TYPE ST_CX_NVDataBlock :
STRUCT
	DataOffs	: UDINT;
	Data		: STRING(2048);
END_STRUCT
END_TYPE

(* stored: Version 1.1.0.1, ProductVersion 3.1.4024.15
   DUT ST_CX_NVDataBlock: Id {52545ff6-35e3-40eb-bc4b-3e33157a43cb} *)
